TYPE ST_St030_Command :
STRUCT
	Command : E_St030_Command;
	Position : INT;
	//IndexX,
	//IndexY	: INT;
END_STRUCT
END_TYPE

(* stored: Version 1.1.0.1
   DUT ST_St030_Command: Id {fbd2d7f3-2a5b-48e4-bb00-6ebb9c76aca9} *)
